DATA_BLOCK "DB_全部电梯"
{ S7_Optimized_Access := 'TRUE' }
VERSION : 0.1
NON_RETAIN
   VAR
      梯数组 : Array[1..3] of "UDT_单梯状态";
   END_VAR


BEGIN

END_DATA_BLOCK

